Fanuc KAREL source: kb00028.KL

-- PROVISIONAL review KL for V770-1; original PC SHA256 41f61f5001041739ac8a8d7728cde8c4cd26d069dcf13779cbbb84c982d215ae
-- Incomplete behavior may be omitted. Consult companion uncertainty JSON. Do not deploy.
PROGRAM KB00028
%NOLOCKGROUP
BEGIN
  -- UNRESOLVED_PC offsets 5-12; opcodes 9D,23
  -- UNRESOLVED_PC offsets 17-26; opcodes 3F,75
  -- UNRESOLVED_PC offsets 31-38; opcodes 9D,23
  -- UNRESOLVED_PC offsets 43-67; opcodes 27,22,22,2A,22,31
  -- UNRESOLVED_PC offsets 72-76; opcodes 7F
END KB00028
